Staubli VAL3: RobotMotion.pgx

program RobotMotion()
begin
  movej(jHome,tTool1,mNomSpeed)
  delay(3)
  while (bBool1)
    call Pick(pPointrx1[nRep])
    nRep=nRep+1

    if nRep==3
      nRep=0
      //bBool1.false
    endIf
    call Place(pPointrx1[nRep])
  endWhile
end
